// TIA Portal V20 export
FUNCTION_BLOCK "Simulation"   // FB194, LAD
// stored: MemoryReserve 100, Namespace Unit1.Em5, SetENOAutomatically false
   VAR_INPUT
      simulation { ExternalAccessible := 'False'; ExternalVisible := 'False'; ExternalWritable := 'False'} : Bool;
   END_VAR
   VAR
      instActuator { ExternalAccessible := 'False'; ExternalVisible := 'False'; ExternalWritable := 'False'} : Array[0..9] of "Simulation_Actuator";
      statDigitalSignal { ExternalAccessible := 'False'; ExternalVisible := 'False'; ExternalWritable := 'False'} : Array[0..9] of Bool;
   END_VAR
   VAR_TEMP   // added for the SCL form of the ladder/FBD networks
      _w1 : Bool;
      _w2 : Bool;
   END_VAR
BEGIN

REGION Network 1: Digital Signal
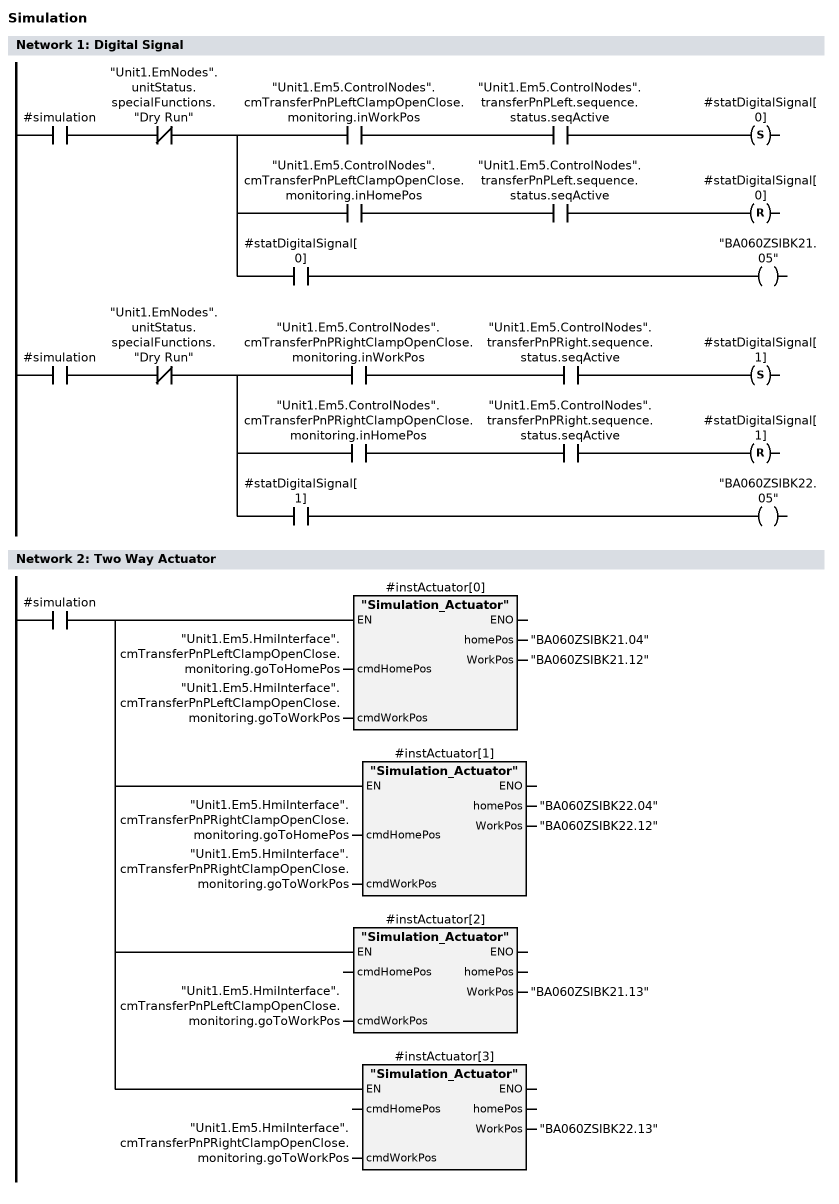
   RUNG wire#powerrail
      Contact( #simulation )
      I_Contact( "Unit1.EmNodes".unitStatus.specialFunctions."Dry Run" )
      wire#w1
      Contact( "Unit1.Em5.ControlNodes".cmTransferPnPLeftClampOpenClose.monitoring.inWorkPos )
      Contact( "Unit1.Em5.ControlNodes".transferPnPLeft.sequence.status.seqActive )
      S_Coil( #statDigitalSignal[0] )
   END_RUNG
   RUNG wire#w1
      Contact( "Unit1.Em5.ControlNodes".cmTransferPnPLeftClampOpenClose.monitoring.inHomePos )
      Contact( "Unit1.Em5.ControlNodes".transferPnPLeft.sequence.status.seqActive )
      R_Coil( #statDigitalSignal[0] )
   END_RUNG
   RUNG wire#w1
      Contact( #statDigitalSignal[0] )
      Coil( "BA060ZSIBK21.05" )
   END_RUNG
   RUNG wire#powerrail
      Contact( #simulation )
      I_Contact( "Unit1.EmNodes".unitStatus.specialFunctions."Dry Run" )
      wire#w2
      Contact( "Unit1.Em5.ControlNodes".cmTransferPnPRightClampOpenClose.monitoring.inWorkPos )
      Contact( "Unit1.Em5.ControlNodes".transferPnPRight.sequence.status.seqActive )
      S_Coil( #statDigitalSignal[1] )
   END_RUNG
   RUNG wire#w2
      Contact( "Unit1.Em5.ControlNodes".cmTransferPnPRightClampOpenClose.monitoring.inHomePos )
      Contact( "Unit1.Em5.ControlNodes".transferPnPRight.sequence.status.seqActive )
      R_Coil( #statDigitalSignal[1] )
   END_RUNG
   RUNG wire#w2
      Contact( #statDigitalSignal[1] )
      Coil( "BA060ZSIBK22.05" )
   END_RUNG
   // the same network as SCL:
   #_w1 := #simulation AND NOT "Unit1.EmNodes".unitStatus.specialFunctions."Dry Run";
   IF #_w1 AND "Unit1.Em5.ControlNodes".cmTransferPnPLeftClampOpenClose.monitoring.inWorkPos AND "Unit1.Em5.ControlNodes".transferPnPLeft.sequence.status.seqActive THEN
       #statDigitalSignal[0] := TRUE;
   END_IF;
   IF #_w1 AND "Unit1.Em5.ControlNodes".cmTransferPnPLeftClampOpenClose.monitoring.inHomePos AND "Unit1.Em5.ControlNodes".transferPnPLeft.sequence.status.seqActive THEN
       #statDigitalSignal[0] := FALSE;
   END_IF;
   "BA060ZSIBK21.05" := #_w1 AND #statDigitalSignal[0];
   #_w2 := #simulation AND NOT "Unit1.EmNodes".unitStatus.specialFunctions."Dry Run";
   IF #_w2 AND "Unit1.Em5.ControlNodes".cmTransferPnPRightClampOpenClose.monitoring.inWorkPos AND "Unit1.Em5.ControlNodes".transferPnPRight.sequence.status.seqActive THEN
       #statDigitalSignal[1] := TRUE;
   END_IF;
   IF #_w2 AND "Unit1.Em5.ControlNodes".cmTransferPnPRightClampOpenClose.monitoring.inHomePos AND "Unit1.Em5.ControlNodes".transferPnPRight.sequence.status.seqActive THEN
       #statDigitalSignal[1] := FALSE;
   END_IF;
   "BA060ZSIBK22.05" := #_w2 AND #statDigitalSignal[1];
END_REGION

REGION Network 2: Two Way Actuator
   RUNG wire#powerrail
      Contact( #simulation )
      wire#w1
      #instActuator[0](cmdHomePos := "Unit1.Em5.HmiInterface".cmTransferPnPLeftClampOpenClose.monitoring.goToHomePos, cmdWorkPos := "Unit1.Em5.HmiInterface".cmTransferPnPLeftClampOpenClose.monitoring.goToWorkPos, homePos => "BA060ZSIBK21.04", WorkPos => "BA060ZSIBK21.12")
   END_RUNG
   RUNG wire#w1
      #instActuator[1](cmdHomePos := "Unit1.Em5.HmiInterface".cmTransferPnPRightClampOpenClose.monitoring.goToHomePos, cmdWorkPos := "Unit1.Em5.HmiInterface".cmTransferPnPRightClampOpenClose.monitoring.goToWorkPos, homePos => "BA060ZSIBK22.04", WorkPos => "BA060ZSIBK22.12")
   END_RUNG
   RUNG wire#w1
      #instActuator[2](cmdHomePos :=, cmdWorkPos := "Unit1.Em5.HmiInterface".cmTransferPnPLeftClampOpenClose.monitoring.goToWorkPos, homePos =>, WorkPos => "BA060ZSIBK21.13")
   END_RUNG
   RUNG wire#w1
      #instActuator[3](cmdHomePos :=, cmdWorkPos := "Unit1.Em5.HmiInterface".cmTransferPnPRightClampOpenClose.monitoring.goToWorkPos, homePos =>, WorkPos => "BA060ZSIBK22.13")
   END_RUNG
   // the same network as SCL:
   IF #simulation THEN
       #instActuator[0](cmdHomePos := "Unit1.Em5.HmiInterface".cmTransferPnPLeftClampOpenClose.monitoring.goToHomePos,   // "Simulation_Actuator"
                        cmdWorkPos := "Unit1.Em5.HmiInterface".cmTransferPnPLeftClampOpenClose.monitoring.goToWorkPos,
                        homePos => "BA060ZSIBK21.04",
                        WorkPos => "BA060ZSIBK21.12");
       #instActuator[1](cmdHomePos := "Unit1.Em5.HmiInterface".cmTransferPnPRightClampOpenClose.monitoring.goToHomePos,   // "Simulation_Actuator"
                        cmdWorkPos := "Unit1.Em5.HmiInterface".cmTransferPnPRightClampOpenClose.monitoring.goToWorkPos,
                        homePos => "BA060ZSIBK22.04",
                        WorkPos => "BA060ZSIBK22.12");
       #instActuator[2](cmdWorkPos := "Unit1.Em5.HmiInterface".cmTransferPnPLeftClampOpenClose.monitoring.goToWorkPos,   // "Simulation_Actuator"
                        WorkPos => "BA060ZSIBK21.13");
       #instActuator[3](cmdWorkPos := "Unit1.Em5.HmiInterface".cmTransferPnPRightClampOpenClose.monitoring.goToWorkPos,   // "Simulation_Actuator"
                        WorkPos => "BA060ZSIBK22.13");
   END_IF;
END_REGION

REGION Network 3 (SCL): homing
   IF #simulation AND "JB_Temp".Test_Homing[5] THEN

       "Unit1.Em5.HmiInterface".cmTransferPnPLeftAxisX.commands.homing :=
       "Unit1.Em5.HmiInterface".cmTransferPnPLeftAxisY.commands.homing :=
       "Unit1.Em5.HmiInterface".cmTransferPnPLeftAxisZ.commands.homing :=
       "Unit1.Em5.HmiInterface".cmTransferPnPRightAxisX.commands.homing :=
       "Unit1.Em5.HmiInterface".cmTransferPnPRightAxisY.commands.homing :=
       "Unit1.Em5.HmiInterface".cmTransferPnPRightAxisZ.commands.homing := true;

       "JB_Temp".Test_Homing[5] := false;
   //    
   END_IF;

   IF #simulation AND "JB_Temp".Test_Homing[20] THEN


       "Unit1.Em5.HmiInterface".cmTransferPnPLeftAxisX.commands.homing :=
       "Unit1.Em5.HmiInterface".cmTransferPnPLeftAxisY.commands.homing :=
       "Unit1.Em5.HmiInterface".cmTransferPnPLeftAxisZ.commands.homing :=
       "Unit1.Em5.HmiInterface".cmTransferPnPRightAxisX.commands.homing :=
       "Unit1.Em5.HmiInterface".cmTransferPnPRightAxisY.commands.homing :=
       "Unit1.Em5.HmiInterface".cmTransferPnPRightAxisZ.commands.homing := false;

   END_IF;
END_REGION
END_FUNCTION_BLOCK
